# EPICS autosave request: dmm7510App/Db/ict_settings.req
# Autosave Request File - ICT
#
# Sample Trigger source
$(P)$(R)SampleTrg-Sel.VAL
# Timer configuration
$(P)$(R)2ndReadDly-SP.VAL
# Digitize Settings
$(P)$(R)SampleCnt-SP.VAL
$(P)$(R)Imped-Sel.VAL
$(P)$(R)Aperture-SP.VAL
$(P)$(R)SampleRate-SP.VAL
# Charge Digitize Range
$(P)$(R)Range-Sel.VAL
$(P)$(R)BCMRange-SP.VAL
# BCM Calibration Settings
$(P)$(R)CalEnbl-Sel.VAL
$(P)$(R)CalCharge-Sel.VAL
# Level Threshold
$(P)$(R)Threshold-SP.VAL
$(P)$(R)HFReject-Sel.VAL
